PROGRAM Motormesswerte
VAR
	v0:LREAL:=0;
	v1:LREAL:=0;
	v2:LREAL:=0;
	
//INPUTS
velocityFromMotor1 AT%I* :LREAL;
velocityFromMotor2 AT%I* :LREAL;
velocityFromMotor3 AT%I* :LREAL;

//OUTPUTS
vXCartesianFromMotors AT%Q*:LREAL;
vYCartesianFromMotors AT%Q*:LREAL;
vthetaCartesianFromMotors AT%Q*:LREAL;

END_VAR

v0:=-velocityFromMotor1;
v1:=-velocityFromMotor2;
v2:=-velocityFromMotor3;

vXCartesianFromMotors:=(v2 - v0) / (2.0 * COS(30.0*PI/180));  //in mm / s
vYCartesianFromMotors:=(v0 - 2.0 * v1 + v2) / 3.0;            //in mm / s
vThetaCartesianFromMotors:=(v0 + v1 + v2) / (3.0 * 135.0);    //in rad / s

END_PROGRAM

(* stored: Version 1.1.0.1, ProductVersion 3.1.4022.3
   POU Motormesswerte: Id {98ef246c-4a5c-421c-b909-7664c31975fe}, SpecialFunc None *)
